TEXTLIST TL_SingleCylinderState_1
  0 = 'Uninitialized'
  10 = 'Initializing'
  20 = 'Ready initialized'
  30 = 'Idle'
  40 = 'Go active'
  50 = 'Go active done'
  60 = 'Go home'
  70 = 'Go home done'
  80 = 'Release'
  90 = 'Release done'
  100 = 'Reset'
  110 = 'Reset done'
  -10 = 'Aborting'
   = ''
END_TEXTLIST

(* stored: Version 1.1.0.1, ProductVersion 3.1.4024.12
   TextList TL_SingleCylinderState_1: Id {fda9eff5-c0f7-407b-81dd-22636138b1cf} *)
